FUNCTION_BLOCK L1_SendCmd (* Basic Function Block Type *)
  (* Standard: 61499-2 *)
  (* Version 0.0, 2015-03-03, EQUEROL, UJI *)
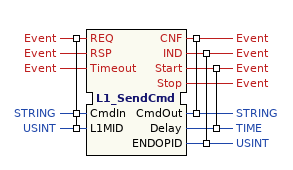
  EVENT_INPUT
    REQ WITH CmdIn, L1MID; (* Normal Execution Request *)
    RSP; (* Cmd reception confirmation *)
    Timeout; (* L0 comm timeout *)
  END_EVENT
  EVENT_OUTPUT
    CNF WITH CmdOut; (* Execution Confirmation *)
    IND WITH ENDOPID; (* Communication Failure indication *)
    Start WITH Delay; (* Start comm timeout *)
    Stop; (* Stop comm timeout *)
  END_EVENT
  VAR_INPUT
    CmdIn : STRING; (* Command string to be sent to the machine *)
    L1MID : USINT; (* Layer 1 multcast identifier *)
  END_VAR
  VAR_OUTPUT
    CmdOut : STRING; (* Command to be sent to the machine *)
    Delay : TIME; (* comm timeout delay *)
    ENDOPID : USINT; (* Indicate upper layer that operation failed *)
  END_VAR
  VAR
    TOCounter : USINT := 0; (* Timeout counter *)
  END_VAR
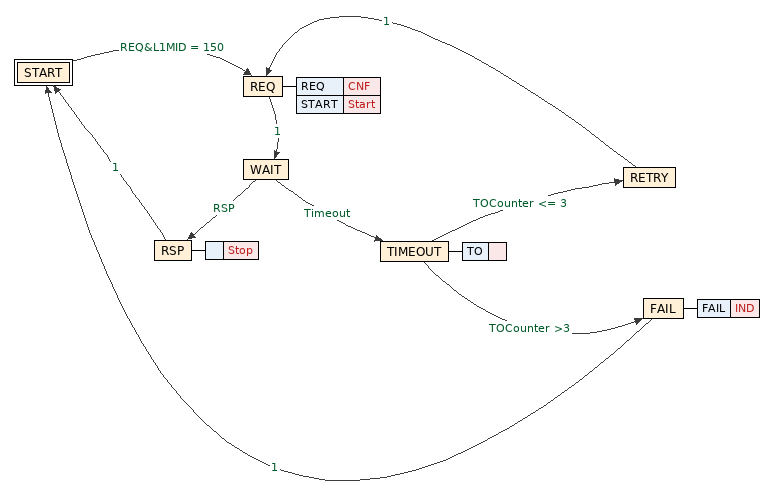
  EC_STATES
    START; (* Initial State *)
    REQ : REQ -> CNF, START -> Start; (* Normal execution *)
    WAIT;
    RSP : -> Stop;
    TIMEOUT : TO;
    RETRY;
    FAIL : FAIL -> IND;
  END_STATES
  EC_TRANSITIONS
    START TO REQ := REQ&L1MID = 150;
    REQ TO WAIT := 1;
    WAIT TO RSP := RSP;
    RSP TO START := 1;
    WAIT TO TIMEOUT := Timeout;
    TIMEOUT TO RETRY := TOCounter <= 3;
    TIMEOUT TO FAIL := TOCounter >3;
    RETRY TO REQ := 1;
    FAIL TO START := 1;
  END_TRANSITIONS
  ALGORITHM REQ IN ST: (* Normally executed algorithm *)
CmdOut := CmdIn;
  END_ALGORITHM
  ALGORITHM START IN ST: (* new algorithm *)
Delay := TIME#1500ms;
  END_ALGORITHM
  ALGORITHM TO IN ST: (* Timeout algo *)
TOCounter := TOCounter + 1;
  END_ALGORITHM
  ALGORITHM RSP IN ST: (* RSP algo *)
TOCounter := 0;
  END_ALGORITHM
  ALGORITHM FAIL IN ST: (* new algorithm *)
TOCounter := 0;
ENDOPID := 1;
  END_ALGORITHM
END_FUNCTION_BLOCK
